PROGRAM MAPPING_in
VAR CONSTANT
//-----------------------------------------------------------------------------------------------------------------
//  Stop! Who approacheth the Bridge of Death must answer me these questions three, ere the other side he see
//-----------------------------------------------------------------------------------------------------------------
{IF defined (AXIS_MAP)}
  {info 'PLC_MOTION_LAYER: AXIS_MAP'}
  bBypassMappingAxis        : BOOL  := FALSE;
{ELSE}
  bBypassMappingAxis        : BOOL  := TRUE;
{END_IF}
//-----------------------------------------------------------------------------------------------------------------
//  What... is your name?
//-----------------------------------------------------------------------------------------------------------------
{IF defined (NCI_MAP)}
  {info 'PLC_MOTION_LAYER: NCI_MAP'}
  bBypassMappingNci         : BOOL  := FALSE;
{ELSE}
  bBypassMappingNci         : BOOL  := TRUE;
{END_IF}
//-----------------------------------------------------------------------------------------------------------------
//  What... is your quest?
//-----------------------------------------------------------------------------------------------------------------
{IF defined (CAM_MAP)}
  {info 'PLC_MOTION_LAYER: CAM_MAP'}
  bBypassMappingCam         : BOOL  := FALSE;
{ELSE}
  bBypassMappingCam         : BOOL  := TRUE;
{END_IF}
//-----------------------------------------------------------------------------------------------------------------
//  What... is the capital of Assyria?
//-----------------------------------------------------------------------------------------------------------------
{IF defined (TRIGGER_MAP)}
  {info 'PLC_MOTION_LAYER: TRIGGER_MAP'}
  bBypassMappingTrigger     : BOOL  := FALSE;
{ELSE}
  bBypassMappingTrigger     : BOOL  := TRUE;
{END_IF}
END_VAR
VAR
  bFirstCycle               : BOOL := TRUE;
//-----------------------------------------------------------------------------------------------------------------
//  Ask me the questions, bridgekeeper. I'm not afraid.
//-----------------------------------------------------------------------------------------------------------------
{IF defined (AXIS_MAP)}
  AxisCtrl                  : U_AXIS_CTRL;
  AxisMoveData              : U_AXIS_MOVE_DATA;
  AxisMotionOptions         : U_AXIS_MOTION_OPTIONS;

  AxisGearInData            : U_AXIS_GEAR_IN;
  AxisHoming                : U_AXIS_HOMING;
  AxisParameterWrt          : U_AXIS_NC_PARAMETER_WRT;
{ELSE}
  AxisCtrl                  : BYTE;
  AxisMoveData              : BYTE;
  AxisMotionOptions         : BYTE;

  AxisGearInData            : BYTE;
  AxisHoming                : BYTE;
  AxisParameterWrt          : BYTE;
{END_IF}
//-----------------------------------------------------------------------------------------------------------------
//  Sir Robin of Camelot.
//-----------------------------------------------------------------------------------------------------------------
{IF defined (NCI_MAP)}
  NciControl                : U_NCI_CTRL;
  NciAxisGroup              : U_NCI_AXIS_ID_GROUP;
  NciRparameters            : U_NCI_R_PARAMETER_I;
{ELSE}
  NciControl                : BYTE;
  NciAxisGroup              : BYTE;
  NciRparameters            : BYTE;
{END_IF}
//-----------------------------------------------------------------------------------------------------------------
//  To seek the Holy Grail.
//-----------------------------------------------------------------------------------------------------------------
{IF defined (CAM_MAP)}
  CamControl                : U_CAM_CTRL;
{ELSE}
  CamControl                : BYTE;
{END_IF}
//-----------------------------------------------------------------------------------------------------------------
//  .....
//-----------------------------------------------------------------------------------------------------------------
{IF defined (TRIGGER_MAP)}
  TriggerControl            : U_TRIGGER_CTRL;
  TouchProbeControl         : U_TOUCH_PROBE_CTRL;
{ELSE}
  //  I don't know that! Auuuuuuuugh!
  TriggerControl            : BYTE;
  TouchProbeControl         : BYTE;
{END_IF}
//-----------------------------------------------------------------------------------------------------------------
//   What... is the air-speed velocity of an unladen swallow?
//-----------------------------------------------------------------------------------------------------------------
  bMappingBlocked           : BOOL;   //  How do know so much about swallows?
//-----------------------------------------------------------------------------------------------------------------
//  - datafield size check
//-----------------------------------------------------------------------------------------------------------------
  szAxisPara,
  szAxisHoming,
  szAxisGearData,
  szAxisMotionOptions,
  szAxisMoveData,
  szAxisCtrl                : ARRAY[1..2] OF UDINT;

  szNciRparameters,
  szNciAxisGroup,
  szNciCtrl                 : ARRAY[1..2] OF UDINT;

  szCamCtrl                 : ARRAY[1..2] OF UDINT;

  szCtrlTouchProbe,
  szCtrlTrigger             : ARRAY[1..2] OF UDINT;
END_VAR

//-----------------------------------------------------------------------------------------------------------------
//  - datafield size check
//-----------------------------------------------------------------------------------------------------------------
IF (bFirstCycle)
THEN
  bFirstCycle             := FALSE;

  szAxisCtrl[1]           := SIZEOF(AxisCtrl);
  szAxisCtrl[2]           := SIZEOF(GVL_AXIS.Ctrl);
  
  szAxisMoveData [1]      := SIZEOF(AxisMoveData);
  szAxisMoveData [2]      := SIZEOF(GVL_AXIS.Data);
  
  szAxisMotionOptions [1] := SIZEOF(AxisMotionOptions);
  szAxisMotionOptions [2] := SIZEOF(GVL_AXIS.MotionOptions);
  
  szAxisGearData [1]      := SIZEOF(AxisGearInData);
  szAxisGearData [2]      := SIZEOF(GVL_AXIS.GearInParameter);
  
  szAxisHoming [1]        := SIZEOF(AxisHoming);
  szAxisHoming [2]        := SIZEOF(GVL_AXIS.HomeParameter);
  
  szAxisPara [1]          := SIZEOF(AxisParameterWrt);
  szAxisPara [2]          := SIZEOF(GVL_AXIS.NcParameterWrt);
 
  szNciRparameters[1]     := SIZEOF(NciRparameters);
  szNciRparameters[2]     := SIZEOF(GVL_NCI.R_ParameterWrite);

  szNciAxisGroup  [1]     := SIZEOF(NciAxisGroup);
  szNciAxisGroup  [2]     := SIZEOF(GVL_NCI.AxisConfig);

  szNciCtrl[1]            := SIZEOF(NciControl);
  szNciCtrl[2]            := SIZEOF(GVL_NCI.ChannelCtrl);
 
  szCamCtrl [1]           := SIZEOF(CamControl);
  szCamCtrl [2]           := SIZEOF(GVL_CAM.Ctrl);
  
  szCtrlTrigger[1]        := SIZEOF(TriggerControl);
  szCtrlTrigger[2]        := SIZEOF(GVL_FUNCTIONS.CtrlTrigger);
  
  szCtrlTouchProbe[1]     := SIZEOF(TouchProbeControl);
  szCtrlTouchProbe[2]     := SIZEOF(GVL_FUNCTIONS.CtrlTouchProbe);
END_IF
//--------------------------------------------------------------------------------------------
//--------------------------------------------------------------------------------------------
//  What do you mean? An African or European swallow?
//--------------------------------------------------------------------------------------------
IF bMappingBlocked
THEN
  RETURN; // Huh? I-- I don't know that. Auuuuuuuugh!
END_IF
//--------------------------------------------------------------------------------------------
//  Well, you have to know these things when you're a king, you know.
//--------------------------------------------------------------------------------------------
//--------------------------------------------------------------------------------------------
//           destination,                         source,                      size
//--------------------------------------------------------------------------------------------
IF NOT bBypassMappingAxis
THEN
  memcpy(ADR(GVL_AXIS.Ctrl),                 ADR(AxisCtrl),             SIZEOF(AxisCTrl));
  memcpy(ADR(GVL_AXIS.Data),                 ADR(AxisMoveData),         SIZEOF(AxisMoveData));
  memcpy(ADR(GVL_AXIS.MotionOptions),        ADR(AxisMotionOptions),    SIZEOF(AxisMotionOptions));

  memcpy(ADR(GVL_AXIS.GearInParameter),      ADR(AxisGearInData),       SIZEOF(AxisGearInData));
  memcpy(ADR(GVL_AXIS.HomeParameter),        ADR(AxisHoming),           SIZEOF(AxisHoming));
  memcpy(ADR(GVL_AXIS.NcParameterWrt),       ADR(AxisParameterWrt),     SIZEOF(AxisParameterWrt));
END_IF
//--------------------------------------------------------------------------------------------
//--------------------------------------------------------------------------------------------
IF NOT bBypassMappingNci
THEN
  memcpy(ADR(GVL_NCI.ChannelCtrl),           ADR(NciControl),           SIZEOF(NciControl));
  memcpy(ADR(GVL_NCI.AxisConfig),            ADR(NciAxisGroup),         SIZEOF(NciAxisGroup));
  memcpy(ADR(GVL_NCI.R_ParameterWrite),      ADR(NciRparameters),       SIZEOF(NciRparameters));
END_IF
//--------------------------------------------------------------------------------------------
//--------------------------------------------------------------------------------------------
IF NOT bBypassMappingCam
THEN
  memcpy(ADR(GVL_CAM.Ctrl),                  ADR(CamControl),           SIZEOF(CamControl));
END_IF
//--------------------------------------------------------------------------------------------
//--------------------------------------------------------------------------------------------
IF NOT bBypassMappingTrigger
THEN
  memcpy(ADR(GVL_FUNCTIONS.CtrlTrigger),     ADR(TriggerControl),       SIZEOF(TriggerControl));
  memcpy(ADR(GVL_FUNCTIONS.CtrlTouchProbe),  ADR(TouchProbeControl),    SIZEOF(TouchProbeControl));
END_IF
//--------------------------------------------------------------------------------------------
//--------------------------------------------------------------------------------------------
//           destination,                         source,                      size
//--------------------------------------------------------------------------------------------

END_PROGRAM

(* stored: Version 1.1.0.1, ProductVersion 3.1.4026.13
   POU MAPPING_in: Id {e84de69b-ba26-07ad-1592-7be68e226b51}, SpecialFunc None *)
